INTERFACE ITF_Component2_HMI_Connector_View EXTENDS ITF_BaseComponent_HMI_Connector_View

END_INTERFACE

(* stored: Version 1.1.0.1
   Itf ITF_Component2_HMI_Connector_View: Id {b91cd31a-3e74-0889-178e-dfc2526a7465} *)
